PROGRAM C12_InfeedConvAddOACData
VAR

	fbAddOACData						: FB_CASE_AddOACDataDBLoop;
	rtrigAddOACData					: R_TRIG;

	nOACFilesRead						: UDINT;
	nReadOACDataFromStructure			: INT;
	nReadOACDataFromFile				: INT;
	nOACFilesFalseRead 				: INT;

	sOACFile							: T_OAC_Filename;
	stLastAddOACData					: ST_OAC_Data;

	fbRestoreOCVData					: FB_CASE_RestoreDataControl;
	sLastResoredOuter					: T_OUTER_Barcode;
END_VAR

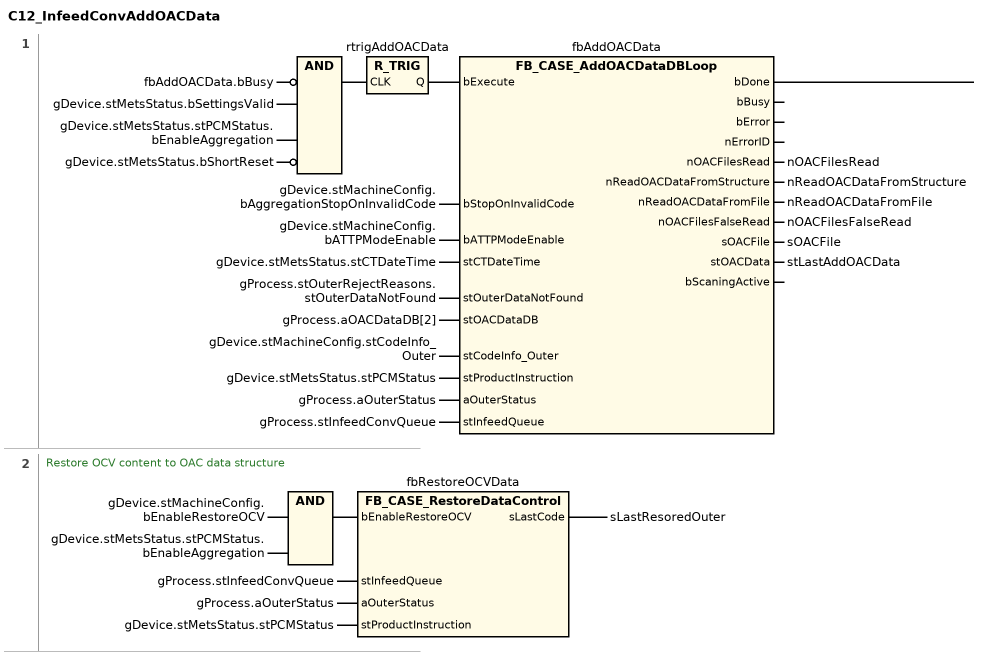
// NETWORK 1
rtrigAddOACData(CLK := NOT fbAddOACData.bBusy AND gDevice.stMetsStatus.bSettingsValid AND gDevice.stMetsStatus.stPCMStatus.bEnableAggregation AND NOT gDevice.stMetsStatus.bShortReset); // R_TRIG
fbAddOACData(
    bExecute := rtrigAddOACData.Q,
    bStopOnInvalidCode := gDevice.stMachineConfig.bAggregationStopOnInvalidCode,
    bATTPModeEnable := gDevice.stMachineConfig.bATTPModeEnable,
    stCTDateTime := gDevice.stMetsStatus.stCTDateTime,
    stOuterDataNotFound := gProcess.stOuterRejectReasons.stOuterDataNotFound,
    stOACDataDB := gProcess.aOACDataDB[2],
    stCodeInfo_Outer := gDevice.stMachineConfig.stCodeInfo_Outer,
    stProductInstruction := gDevice.stMetsStatus.stPCMStatus,
    aOuterStatus := gProcess.aOuterStatus,
    stInfeedQueue := gProcess.stInfeedConvQueue,
    nOACFilesRead => nOACFilesRead,
    nReadOACDataFromStructure => nReadOACDataFromStructure,
    nReadOACDataFromFile => nReadOACDataFromFile,
    nOACFilesFalseRead => nOACFilesFalseRead,
    sOACFile => sOACFile,
    stOACData => stLastAddOACData); // FB_CASE_AddOACDataDBLoop

// NETWORK 2
// Restore OCV content to OAC data structure
fbRestoreOCVData(
    bEnableRestoreOCV := gDevice.stMachineConfig.bEnableRestoreOCV AND gDevice.stMetsStatus.stPCMStatus.bEnableAggregation,
    stInfeedQueue := gProcess.stInfeedConvQueue,
    aOuterStatus := gProcess.aOuterStatus,
    stProductInstruction := gDevice.stMetsStatus.stPCMStatus); // FB_CASE_RestoreDataControl
sLastResoredOuter := fbRestoreOCVData.sLastCode;

END_PROGRAM

(* stored: Version 1.1.0.1
   POU C12_InfeedConvAddOACData: Id {5d75e4ce-291f-4f83-b773-f4b1934943ef}, SpecialFunc None *)
